(* IEC 61131-3 sources: cds-text-sync-reference-project/project-view/CODESYS_Linux_SL/PLC Logic/CI_CD_Application/FunctionBlocks, 4 files *)

(* ---- FB_Counter_UD.st ---- *)
FUNCTION_BLOCK FB_Counter_UD
VAR_INPUT
	xUp : BOOL := FALSE;
	xDown : BOOL := FALSE;
	xReset : BOOL := FALSE;
	uiLimit : UINT := 100;
END_VAR
VAR_OUTPUT
	uiValue : UINT := 0;
	xLimitReached : BOOL := FALSE;
END_VAR
VAR
	_xUpPrev : BOOL := FALSE;
	_xDownPrev : BOOL := FALSE;
END_VAR

// --- implementation ---

// Reset
IF xReset THEN
	uiValue := 0;
	xLimitReached := FALSE;
	_xUpPrev := FALSE;
	_xDownPrev := FALSE;
	RETURN;
END_IF

// Rising edge up
IF xUp AND NOT _xUpPrev THEN
	IF uiValue < uiLimit THEN
		uiValue := uiValue + 1;
	END_IF
END_IF
_xUpPrev := xUp;

// Rising edge down
IF xDown AND NOT _xDownPrev THEN
	IF uiValue > 0 THEN
		uiValue := uiValue - 1;
	END_IF
END_IF
_xDownPrev := xDown;

// Limit detection
xLimitReached := uiValue >= uiLimit;

(* ---- FB_Delay.st ---- *)
FUNCTION_BLOCK FB_Delay
VAR_INPUT
	xTrig : BOOL := FALSE;
	tDelay : TIME := T#1s;
END_VAR
VAR_OUTPUT
	xOut : BOOL := FALSE;
	xElapsed : BOOL := FALSE;
END_VAR
VAR
	_timer : TON;
	_xTrigPrev : BOOL := FALSE;
END_VAR

// --- implementation ---

// Detect rising edge
IF xTrig AND NOT _xTrigPrev THEN
	_timer(IN := TRUE, PT := tDelay);
END_IF
_xTrigPrev := xTrig;

// Run timer
_timer();

xOut := _timer.Q;
xElapsed := _timer.Q AND NOT _xTrigPrev;

(* ---- FB_PulseTrain.st ---- *)
FUNCTION_BLOCK FB_PulseTrain
VAR_INPUT
	xStart : BOOL := FALSE;
	xStop : BOOL := FALSE;
	uiPulseCount : UINT := 10;
	tPeriod : TIME := T#500ms;
END_VAR
VAR_OUTPUT
	xPulse : BOOL := FALSE;
	xBusy : BOOL := FALSE;
	xDone : BOOL := FALSE;
END_VAR
VAR
	_timer : TP;
	_pulseCount : UINT := 0;
	_xStartPrev : BOOL := FALSE;
	_running : BOOL := FALSE;
END_VAR

// --- implementation ---

// Stop
IF xStop THEN
	_running := FALSE;
	_pulseCount := 0;
	xPulse := FALSE;
	xBusy := FALSE;
	xDone := FALSE;
	RETURN;
END_IF

// Start on rising edge
IF xStart AND NOT _xStartPrev THEN
	_running := TRUE;
	_pulseCount := 0;
	xDone := FALSE;
END_IF
_xStartPrev := xStart;

IF _running THEN
	_timer(IN := TRUE, PT := tPeriod);
	xPulse := _timer.Q;

	IF _timer.Q THEN
		_pulseCount := _pulseCount + 1;
		IF _pulseCount >= uiPulseCount THEN
			_running := FALSE;
			xDone := TRUE;
		END_IF
	END_IF

	xBusy := TRUE;
ELSE
	_timer(IN := FALSE);
	xPulse := FALSE;
	xBusy := FALSE;
END_IF

(* ---- FB_TrafficLight.st ---- *)
FUNCTION_BLOCK FB_TrafficLight
VAR_INPUT
	xRun : BOOL := FALSE;
	xReset : BOOL := FALSE;
END_VAR
VAR_OUTPUT
	xRed : BOOL := FALSE;
	xYellow : BOOL := FALSE;
	xGreen : BOOL := FALSE;
	eState : USINT := 0; // 0=Red, 1=RedYellow, 2=Green, 3=Yellow
END_VAR
VAR
	_timer : TON;
	_state : USINT := 0;
	_times : ARRAY[0..3] OF TIME := [T#3s, T#1s, T#3s, T#1s];
	_xRunPrev : BOOL := FALSE;
END_VAR

// --- implementation ---

IF xReset THEN
	_state := 0;
	xRed := FALSE; xYellow := FALSE; xGreen := FALSE;
	eState := 0;
	_timer(IN := FALSE);
	RETURN;
END_IF

// Start on rising edge
IF xRun AND NOT _xRunPrev THEN
	_state := 0;
	_timer(IN := TRUE, PT := _times[0]);
END_IF
_xRunPrev := xRun;

IF NOT xRun THEN
	_timer(IN := FALSE);
	xRed := FALSE; xYellow := FALSE; xGreen := FALSE;
	RETURN;
END_IF

// State machine
_timer();

IF _timer.Q THEN
	_state := (_state + 1) MOD 4;
	_timer(IN := TRUE, PT := _times[_state]);
END_IF

// Output mapping
CASE _state OF
	0: xRed := TRUE;  xYellow := FALSE; xGreen := FALSE;
	1: xRed := TRUE;  xYellow := TRUE;  xGreen := FALSE;
	2: xRed := FALSE; xYellow := FALSE; xGreen := TRUE;
	3: xRed := FALSE; xYellow := TRUE;  xGreen := FALSE;
END_CASE

eState := _state;
